(* CODESYS project XPlanar_Motion.library
   Author: Yuki
   Placeholder: XPlanar_Motion
   Title: XPlanar_Motion
   Version: 1.0
   DefaultNamespace: PM
   Company: Beckhoff

Project tree, tasks and I/O mapping:
  libraries: Tc2_MC2, * (Beckhoff Automation GmbH); Tc2_MC2_Camming, * (Beckhoff Automation GmbH); Tc2_Standard, * (Beckhoff Automation GmbH); Tc2_System, * (Beckhoff Automation GmbH); Tc3_Mc3PlanarMotion, * (Beckhoff Automation GmbH); Tc3_Module, * (Beckhoff Automation GmbH); Tc3_Physics, * (Beckhoff Automation GmbH); Tc3_XPlanarUtility, * (Beckhoff Automation GmbH & Co. KG)
  DUTs/
    data type ST_POSITION
  GVLs/
  POUs/
    General_FB/
      function block FB_StatusExecuteFB [ST]: METH_Busy, METH_CommandAborted, METH_Done, METH_Enter, METH_Error, METH_Execute, METH_Exit, METH_Main, Prop_Busy, Prop_CommandAborted, Prop_Done, Prop_Error, Prop_ErrorID, Prop_Execute
    Interface/
    MotionXPlanar/
      Basic/
        function block FB_Halt [ST]: METH_Busy, METH_Enter, METH_Exit, METH_Main
        function block FB_MoveA [ST]: METH_Busy, METH_Enter, METH_Exit, METH_Main
        function block FB_MoveB [ST]: METH_Busy, METH_Enter, METH_Exit, METH_Main
        function block FB_MoveC [ST]: METH_Busy, METH_Enter, METH_Exit, METH_Main
        function block FB_MoveToPosition [ST]: METH_Busy, METH_Enter, METH_Exit, METH_Main
        function block FB_MoveZ [ST]: METH_Busy, METH_Enter, METH_Exit, METH_Main
      Demo/
        function block FB_Corner [ST]: METH_Busy, METH_Enter, METH_Exit, METH_Main
        function block FB_ExternalSetPoint [ST]: ACT_SetExternalSetPoint, METH_Busy, METH_Enter, METH_Exit, METH_Main
        function block FB_Rotate_C [ST]: METH_Busy, METH_Enter, METH_Exit, METH_Main
        function block FB_Tilt_AB [ST]: METH_Busy, METH_Enter, METH_Exit, METH_Main
        function block FB_UpDown [ST]: METH_Busy, METH_Enter, METH_Exit, METH_Main
    ReadFB/
  VISUs/
*)

// DUTs/ST_POSITION
TYPE ST_POSITION :
STRUCT
	x					: LREAL;
	y					: LREAL;
	z					: LREAL;
	a					: LREAL;
	b					: LREAL;
	c					: LREAL;
END_STRUCT
END_TYPE

// POUs/General_FB/FB_StatusExecuteFB
 {attribute 'hide'}
FUNCTION_BLOCK ABSTRACT FB_StatusExecuteFB
VAR_INPUT
END_VAR
VAR_OUTPUT
END_VAR
VAR
	bExecute						: BOOL;
	bBusy							: BOOL;
	bCommandAborted					: BOOL;
	bDone							: BOOL;
	bError							: BOOL;
	udiErrorID						: UDINT;
END_VAR

//{warning 'add method implementation '}
METHOD ABSTRACT METH_Busy : BOOL
END_METHOD

//{warning 'add method implementation '}
METHOD PROTECTED METH_CommandAborted : BOOL
Prop_CommandAborted := TRUE;
Prop_Busy := FALSE;
END_METHOD

//{warning 'add method implementation '}
METHOD PROTECTED METH_Done : BOOL
Prop_Done := TRUE;
Prop_Busy := FALSE;
END_METHOD

METHOD ABSTRACT METH_Enter : BOOL
VAR_INPUT
END_VAR
END_METHOD

//{warning 'add method implementation '}
METHOD PROTECTED METH_Error : BOOL
Prop_Error := TRUE;
Prop_Busy := FALSE;
END_METHOD

//{warning 'add method implementation '}
METHOD PROTECTED METH_Execute : BOOL
Prop_Execute := TRUE;
Prop_Busy := TRUE;
END_METHOD

METHOD ABSTRACT METH_Exit : BOOL
VAR_INPUT
END_VAR
END_METHOD

METHOD ABSTRACT METH_Main : BOOL
VAR_INPUT
END_VAR
END_METHOD

{warning 'add property implementation'}
PROPERTY Prop_Busy : BOOL
GET
Prop_Busy := bBusy;
END_GET
SET
bBusy := Prop_Busy;
END_SET
END_PROPERTY

{warning 'add property implementation'}
PROPERTY Prop_CommandAborted : BOOL
GET
Prop_CommandAborted := bCommandAborted;
END_GET
SET
bCommandAborted := Prop_CommandAborted;
END_SET
END_PROPERTY

{warning 'add property implementation'}
PROPERTY Prop_Done : BOOL
GET
Prop_Done := bDone;
END_GET
SET
bDone := Prop_Done;
END_SET
END_PROPERTY

{warning 'add property implementation'}
PROPERTY Prop_Error : BOOL
GET
Prop_Error := bError;
END_GET
SET
bError := Prop_Error;
END_SET
END_PROPERTY

{warning 'add property implementation'}
PROPERTY Prop_ErrorID : UDINT
GET
Prop_ErrorID := udiErrorID;
END_GET
SET
udiErrorID := Prop_ErrorID;
END_SET
END_PROPERTY

{warning 'add property implementation'}
PROPERTY Prop_Execute : BOOL
GET
Prop_Execute := bExecute;
END_GET
SET
bExecute := Prop_Execute;
END_SET
END_PROPERTY

END_FUNCTION_BLOCK

// POUs/MotionXPlanar/Basic/FB_Halt
FUNCTION_BLOCK FB_Halt EXTENDS FB_StatusExecuteFB
VAR_IN_OUT
	fbMover								: MC_PlanarMover;
END_VAR
VAR_INPUT
	Execute								: BOOL;
	Velocity							: LREAL;
	Acceleration						: LREAL;
	Deceleration						: LREAL;
	Jerk								: LREAL;
END_VAR
VAR_OUTPUT
	Done								: BOOL;
	Busy								: BOOL;
	CommandAborted						: BOOL;
	Error								: BOOL;
	ErrorID								: UDINT;
END_VAR
VAR
	uiState								: UINT;
	//Input 内部変数
	lrVelocity							: LREAL;
	lrAcceleration						: LREAL;
	lrDeceleration						: LREAL;
	lrJerk								: LREAL;
	
	//ローカル
	fbFB_Mover							: MC_PlanarFeedback;
	fbConstraint						: DynamicConstraint_PathXY;
END_VAR

Prop_Execute := Execute;
METH_Main();
fbFB_Mover.Update();

Busy := bBusy;
Done := bDone;
CommandAborted := bCommandAborted;
Error := bError;
ErrorID := udiErrorID;

//{error 'add method implementation or delete method to use base implementation'}
METHOD METH_Busy : BOOL
IF fbFB_Mover.Error THEN
	METH_Error();
	Prop_ErrorID := fbFB_Mover.ErrorId; //Moverがエラー
	RETURN;
END_IF
IF THIS^.fbMover.MCTOPLC.STD.State = MC_PLANAR_STATE.Error THEN
	METH_Error();
	Prop_ErrorID := 1; //Moverがエラー
	RETURN;
END_IF
IF fbFB_Mover.Aborted THEN
	METH_CommandAborted();
	RETURN;
END_IF

CASE THIS^.uiState OF
	0:
	fbConstraint.SetValuesVADJ(V:= THIS^.lrVelocity, A:= THIS^.lrAcceleration, D:= THIS^.lrDeceleration, J:= THIS^.lrJerk);
	THIS^.fbMover.Halt(
		commandFeedback:= THIS^.fbFB_Mover, 
		constraint:= fbConstraint);

	THIS^.uiState := 10;	
	
	10:
	IF fbFB_Mover.Done THEN
		THIS^.uiState := 16#FFFF;	
	END_IF
	
	16#FFFF:
	METH_Done();
END_CASE
END_METHOD

//{error 'add method implementation or delete method to use base implementation'}
METHOD METH_Enter : BOOL
//Input 内部変数に移す
lrVelocity := Velocity;
lrAcceleration := Acceleration;
lrDeceleration := Deceleration;
lrJerk := Jerk;
END_METHOD

//{error 'add method implementation or delete method to use base implementation'}
METHOD METH_Exit : BOOL
Prop_Done := FALSE;
Prop_Busy := FALSE;
Prop_CommandAborted := FALSE;
Prop_Error := FALSE;
Prop_ErrorID := 0;

// 内部変数をリフレッシュする
uiState := 0;
lrVelocity := 0;
lrAcceleration := 0;
lrDeceleration := 0;
lrJerk := 0;
END_METHOD

//{error 'add method implementation or delete method to use base implementation'}
METHOD METH_Main : BOOL
//Doneに遷移
IF SUPER^.bDone AND SUPER^.bExecute THEN
	METH_Done();
	RETURN;
END_IF
//Errorに遷移
IF SUPER^.bError AND SUPER^.bExecute THEN
	METH_Error();
	RETURN;
END_IF
//CommandAbortedに遷移
IF SUPER^.bCommandAborted AND SUPER^.bExecute THEN
	METH_CommandAborted();
	RETURN;
END_IF
//FBをリフレッシュ
//状態がDone, Error, CommandAborted時に Execute FALSE で遷移
IF (SUPER^.bDone OR SUPER^.bError OR SUPER^.bCommandAborted) AND NOT SUPER^.bExecute THEN
	METH_Exit();
	RETURN;
END_IF

//実行開始
IF SUPER^.bExecute AND NOT SUPER^.bBusy THEN
	METH_Execute();
	METH_Enter();
END_IF
//実行中
IF SUPER^.bBusy THEN
	METH_Busy();
END_IF
END_METHOD

END_FUNCTION_BLOCK

// POUs/MotionXPlanar/Basic/FB_MoveA
FUNCTION_BLOCK FB_MoveA EXTENDS FB_StatusExecuteFB
VAR_IN_OUT
	fbMover								: MC_PlanarMover;
END_VAR
VAR_INPUT
	Execute								: BOOL;
	Position							: ST_POSITION;
	Velocity							: LREAL;
	Acceleration						: LREAL;
	Deceleration						: LREAL;
	Jerk								: LREAL;
END_VAR
VAR_OUTPUT
	Done								: BOOL;
	Busy								: BOOL;
	CommandAborted						: BOOL;
	Error								: BOOL;
	ErrorID								: UDINT;
END_VAR
VAR
	uiState								: UINT;
	//Input 内部変数
	dutPosition							: ST_POSITION;
	lrVelocity							: LREAL;
	lrAcceleration						: LREAL;
	lrDeceleration						: LREAL;
	lrJerk								: LREAL;
	
	//ローカル
	fbFB_Mover							: MC_PlanarFeedback;
	fbConstraint						: DynamicConstraint_PathXY;
END_VAR

Prop_Execute := Execute;
METH_Main();

fbFB_Mover.Update();

Busy := bBusy;
Done := bDone;
CommandAborted := bCommandAborted;
Error := bError;
ErrorID := udiErrorID;

//{error 'add method implementation or delete method to use base implementation'}
METHOD METH_Busy : BOOL
{warning disable C0371}
{warning restore C0371}
IF fbFB_Mover.Error THEN
	METH_Error();
	Prop_ErrorID := fbFB_Mover.ErrorId; //Moverがエラー
	RETURN;
END_IF
IF THIS^.fbMover.MCTOPLC.STD.State = MC_PLANAR_STATE.Error THEN
	METH_Error();
	Prop_ErrorID := 1; //Moverがエラー
	RETURN;
END_IF
IF fbFB_Mover.Aborted THEN
	METH_CommandAborted();
	RETURN;
END_IF

CASE THIS^.uiState OF
	0:
	fbConstraint.SetValuesVADJ(V:= THIS^.lrVelocity, A:= THIS^.lrAcceleration, D:= THIS^.lrDeceleration, J:= THIS^.lrJerk);
	THIS^.fbMover.MoveA(
		commandFeedback:= THIS^.fbFB_Mover, 
		targetPosition:= dutPosition.a, 
		constraint:= fbConstraint);

	THIS^.uiState := 10;	
	
	10:
	IF fbFB_Mover.Done THEN
		THIS^.uiState := 16#FFFF;	
	END_IF
	
	16#FFFF:
	METH_Done();
END_CASE
END_METHOD

//{error 'add method implementation or delete method to use base implementation'}
METHOD METH_Enter : BOOL
//Input 内部変数に移す
dutPosition := Position;
lrVelocity := Velocity;
lrAcceleration := Acceleration;
lrDeceleration := Deceleration;
lrJerk := Jerk;
END_METHOD

//{error 'add method implementation or delete method to use base implementation'}
METHOD METH_Exit : BOOL
Prop_Done := FALSE;
Prop_Busy := FALSE;
Prop_CommandAborted := FALSE;
Prop_Error := FALSE;
Prop_ErrorID := 0;

// 内部変数をリフレッシュする
uiState := 0;
lrVelocity := 0;
lrAcceleration := 0;
lrDeceleration := 0;
lrJerk := 0;
END_METHOD

//{error 'add method implementation or delete method to use base implementation'}
METHOD METH_Main : BOOL
//Doneに遷移
IF SUPER^.bDone AND SUPER^.bExecute THEN
	METH_Done();
	RETURN;
END_IF
//Errorに遷移
IF SUPER^.bError AND SUPER^.bExecute THEN
	METH_Error();
	RETURN;
END_IF
//CommandAbortedに遷移
IF SUPER^.bCommandAborted AND SUPER^.bExecute THEN
	METH_CommandAborted();
	RETURN;
END_IF
//FBをリフレッシュ
//状態がDone, Error, CommandAborted時に Execute FALSE で遷移
IF (SUPER^.bDone OR SUPER^.bError OR SUPER^.bCommandAborted) AND NOT SUPER^.bExecute THEN
	METH_Exit();
	RETURN;
END_IF

//実行開始
IF SUPER^.bExecute AND NOT SUPER^.bBusy THEN
	METH_Execute();
	METH_Enter();
END_IF
//実行中
IF SUPER^.bBusy THEN
	METH_Busy();
END_IF
END_METHOD

END_FUNCTION_BLOCK

// POUs/MotionXPlanar/Basic/FB_MoveB
FUNCTION_BLOCK FB_MoveB EXTENDS FB_StatusExecuteFB
VAR_IN_OUT
	fbMover								: MC_PlanarMover;
END_VAR
VAR_INPUT
	Execute								: BOOL;
	Position							: ST_POSITION;
	Velocity							: LREAL;
	Acceleration						: LREAL;
	Deceleration						: LREAL;
	Jerk								: LREAL;
END_VAR
VAR_OUTPUT
	Done								: BOOL;
	Busy								: BOOL;
	CommandAborted						: BOOL;
	Error								: BOOL;
	ErrorID								: UDINT;
END_VAR
VAR
	uiState								: UINT;
	//Input 内部変数
	dutPosition							: ST_POSITION;
	lrVelocity							: LREAL;
	lrAcceleration						: LREAL;
	lrDeceleration						: LREAL;
	lrJerk								: LREAL;
	
	//ローカル
	fbFB_Mover							: MC_PlanarFeedback;
	fbConstraint						: DynamicConstraint_PathXY;
END_VAR

Prop_Execute := Execute;
METH_Main();

fbFB_Mover.Update();

Busy := bBusy;
Done := bDone;
CommandAborted := bCommandAborted;
Error := bError;
ErrorID := udiErrorID;

//{error 'add method implementation or delete method to use base implementation'}
METHOD METH_Busy : BOOL
{warning disable C0371}
{warning restore C0371}
IF fbFB_Mover.Error THEN
	METH_Error();
	Prop_ErrorID := fbFB_Mover.ErrorId; //Moverがエラー
	RETURN;
END_IF
IF THIS^.fbMover.MCTOPLC.STD.State = MC_PLANAR_STATE.Error THEN
	METH_Error();
	Prop_ErrorID := 1; //Moverがエラー
	RETURN;
END_IF
IF fbFB_Mover.Aborted THEN
	METH_CommandAborted();
	RETURN;
END_IF

CASE THIS^.uiState OF
	0:
	fbConstraint.SetValuesVADJ(V:= THIS^.lrVelocity, A:= THIS^.lrAcceleration, D:= THIS^.lrDeceleration, J:= THIS^.lrJerk);
	THIS^.fbMover.MoveB(
		commandFeedback:= THIS^.fbFB_Mover, 
		targetPosition:= dutPosition.b, 
		constraint:= fbConstraint);

	THIS^.uiState := 10;	
	
	10:
	IF fbFB_Mover.Done THEN
		THIS^.uiState := 16#FFFF;	
	END_IF
	
	16#FFFF:
	METH_Done();
END_CASE
END_METHOD

//{error 'add method implementation or delete method to use base implementation'}
METHOD METH_Enter : BOOL
//Input 内部変数に移す
dutPosition := Position;
lrVelocity := Velocity;
lrAcceleration := Acceleration;
lrDeceleration := Deceleration;
lrJerk := Jerk;
END_METHOD

//{error 'add method implementation or delete method to use base implementation'}
METHOD METH_Exit : BOOL
Prop_Done := FALSE;
Prop_Busy := FALSE;
Prop_CommandAborted := FALSE;
Prop_Error := FALSE;
Prop_ErrorID := 0;

// 内部変数をリフレッシュする
uiState := 0;
lrVelocity := 0;
lrAcceleration := 0;
lrDeceleration := 0;
lrJerk := 0;
END_METHOD

//{error 'add method implementation or delete method to use base implementation'}
METHOD METH_Main : BOOL
//Doneに遷移
IF SUPER^.bDone AND SUPER^.bExecute THEN
	METH_Done();
	RETURN;
END_IF
//Errorに遷移
IF SUPER^.bError AND SUPER^.bExecute THEN
	METH_Error();
	RETURN;
END_IF
//CommandAbortedに遷移
IF SUPER^.bCommandAborted AND SUPER^.bExecute THEN
	METH_CommandAborted();
	RETURN;
END_IF
//FBをリフレッシュ
//状態がDone, Error, CommandAborted時に Execute FALSE で遷移
IF (SUPER^.bDone OR SUPER^.bError OR SUPER^.bCommandAborted) AND NOT SUPER^.bExecute THEN
	METH_Exit();
	RETURN;
END_IF

//実行開始
IF SUPER^.bExecute AND NOT SUPER^.bBusy THEN
	METH_Execute();
	METH_Enter();
END_IF
//実行中
IF SUPER^.bBusy THEN
	METH_Busy();
END_IF
END_METHOD

END_FUNCTION_BLOCK

// POUs/MotionXPlanar/Basic/FB_MoveC
FUNCTION_BLOCK FB_MoveC EXTENDS FB_StatusExecuteFB
VAR_IN_OUT
	fbMover								: MC_PlanarMover;
END_VAR
VAR_INPUT
	Execute								: BOOL;
	Position							: ST_POSITION;
	Velocity							: LREAL;
	Acceleration						: LREAL;
	Deceleration						: LREAL;
	Jerk								: LREAL;
END_VAR
VAR_OUTPUT
	Done								: BOOL;
	Busy								: BOOL;
	CommandAborted						: BOOL;
	Error								: BOOL;
	ErrorID								: UDINT;
END_VAR
VAR
	uiState								: UINT;
	//Input 内部変数
	dutPosition							: ST_POSITION;
	lrVelocity							: LREAL;
	lrAcceleration						: LREAL;
	lrDeceleration						: LREAL;
	lrJerk								: LREAL;
	
	//ローカル
	fbFB_Mover							: MC_PlanarFeedback;
	fbConstraint						: DynamicConstraint_PathXY;
	stMoveCOptions						: ST_MoveCOptions;
END_VAR

Prop_Execute := Execute;
METH_Main();

fbFB_Mover.Update();

Busy := bBusy;
Done := bDone;
CommandAborted := bCommandAborted;
Error := bError;
ErrorID := udiErrorID;

//{error 'add method implementation or delete method to use base implementation'}
METHOD METH_Busy : BOOL
IF fbFB_Mover.Error THEN
	METH_Error();
	Prop_ErrorID := fbFB_Mover.ErrorId; //Moverがエラー
	RETURN;
END_IF
IF THIS^.fbMover.MCTOPLC.STD.State = MC_PLANAR_STATE.Error THEN
	METH_Error();
	Prop_ErrorID := 1; //Moverがエラー
	RETURN;
END_IF
IF fbFB_Mover.Aborted THEN
	METH_CommandAborted();
	RETURN;
END_IF

CASE THIS^.uiState OF
	0:
	fbConstraint.SetValuesVADJ(V:= THIS^.lrVelocity, A:= THIS^.lrAcceleration, D:= THIS^.lrDeceleration, J:= THIS^.lrJerk);
	//ノンモジュロ設定有効
	stMoveCOptions.direction := Tc3_Mc3PlanarMotion.MC_DIRECTION.mcDirectionNonModulo;
	THIS^.fbMover.MoveC(
		commandFeedback:= THIS^.fbFB_Mover, 
		targetPosition:= dutPosition.c, 
		constraint:= fbConstraint, 
		options:= stMoveCOptions);
	THIS^.uiState := 10;	
	
	10:
	IF fbFB_Mover.Done THEN
		THIS^.uiState := 16#FFFF;	
	END_IF
	
	16#FFFF:
	METH_Done();
END_CASE
END_METHOD

//{error 'add method implementation or delete method to use base implementation'}
METHOD METH_Enter : BOOL
//Input 内部変数に移す
dutPosition := Position;
lrVelocity := Velocity;
lrAcceleration := Acceleration;
lrDeceleration := Deceleration;
lrJerk := Jerk;
END_METHOD

//{error 'add method implementation or delete method to use base implementation'}
METHOD METH_Exit : BOOL
Prop_Done := FALSE;
Prop_Busy := FALSE;
Prop_CommandAborted := FALSE;
Prop_Error := FALSE;
Prop_ErrorID := 0;

// 内部変数をリフレッシュする
uiState := 0;
lrVelocity := 0;
lrAcceleration := 0;
lrDeceleration := 0;
lrJerk := 0;
END_METHOD

//{error 'add method implementation or delete method to use base implementation'}
METHOD METH_Main : BOOL
//Doneに遷移
IF SUPER^.bDone AND SUPER^.bExecute THEN
	METH_Done();
	RETURN;
END_IF
//Errorに遷移
IF SUPER^.bError AND SUPER^.bExecute THEN
	METH_Error();
	RETURN;
END_IF
//CommandAbortedに遷移
IF SUPER^.bCommandAborted AND SUPER^.bExecute THEN
	METH_CommandAborted();
	RETURN;
END_IF
//FBをリフレッシュ
//状態がDone, Error, CommandAborted時に Execute FALSE で遷移
IF (SUPER^.bDone OR SUPER^.bError OR SUPER^.bCommandAborted) AND NOT SUPER^.bExecute THEN
	METH_Exit();
	RETURN;
END_IF

//実行開始
IF SUPER^.bExecute AND NOT SUPER^.bBusy THEN
	METH_Execute();
	METH_Enter();
END_IF
//実行中
IF SUPER^.bBusy THEN
	METH_Busy();
END_IF
END_METHOD

END_FUNCTION_BLOCK

// POUs/MotionXPlanar/Basic/FB_MoveToPosition
FUNCTION_BLOCK FB_MoveToPosition EXTENDS FB_StatusExecuteFB
VAR_IN_OUT
	fbMover								: MC_PlanarMover;
END_VAR
VAR_INPUT
	Execute								: BOOL;
	Position							: ST_POSITION;
	Velocity							: LREAL;
	Acceleration						: LREAL;
	Deceleration						: LREAL;
	Jerk								: LREAL;
END_VAR
VAR_OUTPUT
	Done								: BOOL;
	Busy								: BOOL;
	CommandAborted						: BOOL;
	Error								: BOOL;
	ErrorID								: UDINT;
END_VAR
VAR
	uiState								: UINT;
	//Input 内部変数
	xycPosition							: PositionXYC;
	dutPosition							: ST_POSITION;
	lrVelocity							: LREAL;
	lrAcceleration						: LREAL;
	lrDeceleration						: LREAL;
	lrJerk								: LREAL;
	
	//ローカル
	fbFB_Mover							: MC_PlanarFeedback;
	fbConstraint						: DynamicConstraint_PathXY;
END_VAR

Prop_Execute := Execute;
METH_Main();

fbFB_Mover.Update();

Busy := bBusy;
Done := bDone;
CommandAborted := bCommandAborted;
Error := bError;
ErrorID := udiErrorID;

//{warning 'add method implementation '}
//実行動作
METHOD METH_Busy : BOOL
IF fbFB_Mover.Error THEN
	METH_Error();
	Prop_ErrorID := fbFB_Mover.ErrorId; //Moverがエラー
	RETURN;
END_IF
IF THIS^.fbMover.MCTOPLC.STD.State = MC_PLANAR_STATE.Error THEN
	METH_Error();
	Prop_ErrorID := 1; //Moverがエラー
	RETURN;
END_IF
IF fbFB_Mover.Aborted THEN
	METH_CommandAborted();
	RETURN;
END_IF

CASE THIS^.uiState OF
	0:
	xycPosition.SetValuesXYC(x:= dutPosition.x, y:= dutPosition.y, c:= 0);
	fbConstraint.SetValuesVADJ(V:= THIS^.lrVelocity, A:= THIS^.lrAcceleration, D:= THIS^.lrDeceleration, J:= THIS^.lrJerk);
	THIS^.fbMover.MoveToPosition(
		commandFeedback:= THIS^.fbFB_Mover, 
		targetPosition:= xycPosition, 
		constraint:= fbConstraint, 
		options:= 0);
	THIS^.uiState := 10;
		
	10:
	IF fbFB_Mover.Done THEN
		THIS^.uiState := 16#FFFF;
	END_IF
	
	16#FFFF:
	METH_Done();
END_CASE
END_METHOD

METHOD METH_Enter : BOOL
VAR_INPUT
END_VAR
//Input 内部変数に移す
dutPosition := Position;
lrVelocity := Velocity;
lrAcceleration := Acceleration;
lrDeceleration := Deceleration;
lrJerk := Jerk;
END_METHOD

METHOD METH_Exit : BOOL
VAR_INPUT
END_VAR
Prop_Done := FALSE;
Prop_Busy := FALSE;
Prop_CommandAborted := FALSE;
Prop_Error := FALSE;
Prop_ErrorID := 0;

// 内部変数をリフレッシュする
uiState := 0;
xycPosition.SetValuesXYC(0,0,0);
lrVelocity := 0;
lrAcceleration := 0;
lrDeceleration := 0;
lrJerk := 0;
END_METHOD

METHOD METH_Main : BOOL
VAR_INPUT
END_VAR
//Doneに遷移
IF SUPER^.bDone AND SUPER^.bExecute THEN
	METH_Done();
	RETURN;
END_IF
//Errorに遷移
IF SUPER^.bError AND SUPER^.bExecute THEN
	METH_Error();
	RETURN;
END_IF
//CommandAbortedに遷移
IF SUPER^.bCommandAborted AND SUPER^.bExecute THEN
	METH_CommandAborted();
	RETURN;
END_IF
//FBをリフレッシュ
//状態がDone, Error, CommandAborted時に Execute FALSE で遷移
IF (SUPER^.bDone OR SUPER^.bError OR SUPER^.bCommandAborted) AND NOT SUPER^.bExecute THEN
	METH_Exit();
	RETURN;
END_IF

//実行開始
IF SUPER^.bExecute AND NOT SUPER^.bBusy THEN
	METH_Execute();
	METH_Enter();
END_IF
//実行中
IF SUPER^.bBusy THEN
	METH_Busy();
END_IF
END_METHOD

END_FUNCTION_BLOCK

// POUs/MotionXPlanar/Basic/FB_MoveZ
FUNCTION_BLOCK FB_MoveZ EXTENDS FB_StatusExecuteFB
VAR_IN_OUT
	fbMover								: MC_PlanarMover;
END_VAR
VAR_INPUT
	Execute								: BOOL;
	Position							: ST_POSITION;
	Velocity							: LREAL;
	Acceleration						: LREAL;
	Deceleration						: LREAL;
	Jerk								: LREAL;
END_VAR
VAR_OUTPUT
	Done								: BOOL;
	Busy								: BOOL;
	CommandAborted						: BOOL;
	Error								: BOOL;
	ErrorID								: UDINT;
END_VAR
VAR
	uiState								: UINT;
	//Input 内部変数
	dutPosition							: ST_POSITION;
	lrVelocity							: LREAL;
	lrAcceleration						: LREAL;
	lrDeceleration						: LREAL;
	lrJerk								: LREAL;
	
	//ローカル
	fbFB_Mover							: MC_PlanarFeedback;
	fbConstraint						: DynamicConstraint_PathXY;
END_VAR

Prop_Execute := Execute;
METH_Main();

fbFB_Mover.Update();

Busy := bBusy;
Done := bDone;
CommandAborted := bCommandAborted;
Error := bError;
ErrorID := udiErrorID;

//{error 'add method implementation or delete method to use base implementation'}
METHOD METH_Busy : BOOL
IF fbFB_Mover.Error THEN
	METH_Error();
	Prop_ErrorID := fbFB_Mover.ErrorId; //Moverがエラー
	RETURN;
END_IF
IF THIS^.fbMover.MCTOPLC.STD.State = MC_PLANAR_STATE.Error THEN
	METH_Error();
	Prop_ErrorID := 1; //Moverがエラー
	RETURN;
END_IF
IF fbFB_Mover.Aborted THEN
	METH_CommandAborted();
	RETURN;
END_IF

CASE THIS^.uiState OF
	0:
	fbConstraint.SetValuesVADJ(V:= THIS^.lrVelocity, A:= THIS^.lrAcceleration, D:= THIS^.lrDeceleration, J:= THIS^.lrJerk);
	THIS^.fbMover.MoveZ(
		commandFeedback:= THIS^.fbFB_Mover, 
		targetPosition:= dutPosition.z, 
		constraint:= fbConstraint);

	THIS^.uiState := 10;	
	
	10:
	IF fbFB_Mover.Done THEN
		THIS^.uiState := 16#FFFF;	
	END_IF
	
	16#FFFF:
	METH_Done();
END_CASE
END_METHOD

//{error 'add method implementation or delete method to use base implementation'}
METHOD METH_Enter : BOOL
//Input 内部変数に移す
dutPosition := Position;
lrVelocity := Velocity;
lrAcceleration := Acceleration;
lrDeceleration := Deceleration;
lrJerk := Jerk;
END_METHOD

//{error 'add method implementation or delete method to use base implementation'}
METHOD METH_Exit : BOOL
Prop_Done := FALSE;
Prop_Busy := FALSE;
Prop_CommandAborted := FALSE;
Prop_Error := FALSE;
Prop_ErrorID := 0;

// 内部変数をリフレッシュする
uiState := 0;
lrVelocity := 0;
lrAcceleration := 0;
lrDeceleration := 0;
lrJerk := 0;
END_METHOD

//{error 'add method implementation or delete method to use base implementation'}
METHOD METH_Main : BOOL
//Doneに遷移
IF SUPER^.bDone AND SUPER^.bExecute THEN
	METH_Done();
	RETURN;
END_IF
//Errorに遷移
IF SUPER^.bError AND SUPER^.bExecute THEN
	METH_Error();
	RETURN;
END_IF
//CommandAbortedに遷移
IF SUPER^.bCommandAborted AND SUPER^.bExecute THEN
	METH_CommandAborted();
	RETURN;
END_IF
//FBをリフレッシュ
//状態がDone, Error, CommandAborted時に Execute FALSE で遷移
IF (SUPER^.bDone OR SUPER^.bError OR SUPER^.bCommandAborted) AND NOT SUPER^.bExecute THEN
	METH_Exit();
	RETURN;
END_IF

//実行開始
IF SUPER^.bExecute AND NOT SUPER^.bBusy THEN
	METH_Execute();
	METH_Enter();
END_IF
//実行中
IF SUPER^.bBusy THEN
	METH_Busy();
END_IF
END_METHOD

END_FUNCTION_BLOCK

// POUs/MotionXPlanar/Demo/FB_Corner
FUNCTION_BLOCK FINAL FB_Corner EXTENDS FB_StatusExecuteFB
VAR_IN_OUT
	fbMover								: MC_PlanarMover;
END_VAR
VAR_INPUT
	Execute								: BOOL;
	Position							: ARRAY [0..3] OF ST_POSITION;
	Velocity							: LREAL;
	Acceleration						: LREAL;
	Deceleration						: LREAL;
	Jerk								: LREAL;
END_VAR
VAR_OUTPUT
	Done								: BOOL;
	Busy								: BOOL;
	CommandAborted						: BOOL;
	Error								: BOOL;
	ErrorID								: UDINT;
END_VAR
VAR
	uiState								: UINT;
	//Input 内部変数
	xycPosition							: PositionXYC;
	adutPosition							: ARRAY [0..3] OF ST_POSITION;
	lrVelocity							: LREAL;
	lrAcceleration						: LREAL;
	lrDeceleration						: LREAL;
	lrJerk								: LREAL;
	
	//ローカル
	fbFB_Mover							: MC_PlanarFeedback;
	fbMoveToPosition					: FB_MoveToPosition;
END_VAR

Prop_Execute := Execute;
METH_Main();

fbFB_Mover.Update();

Busy := bBusy;
Done := bDone;
CommandAborted := bCommandAborted;
Error := bError;
ErrorID := udiErrorID;

//{error 'add method implementation or delete method to use base implementation'}
METHOD METH_Busy : BOOL
{warning disable C0371}
{warning restore C0371}
IF fbFB_Mover.Error THEN
	METH_Error();
	Prop_ErrorID := fbFB_Mover.ErrorId; //Moverがエラー
	RETURN;
END_IF
IF THIS^.fbMover.MCTOPLC.STD.State = MC_PLANAR_STATE.Error THEN
	METH_Error();
	Prop_ErrorID := 1; //Moverがエラー
	RETURN;
END_IF
IF fbFB_Mover.Aborted THEN
	METH_CommandAborted();
	RETURN;
END_IF

CASE THIS^.uiState OF
	0:
	//配列0に移動
	fbMoveToPosition(
		fbMover:= THIS^.fbMover, 
		Execute:= TRUE, 
		Position:= adutPosition[0], 
		Velocity:= THIS^.lrVelocity, 
		Acceleration:= THIS^.lrAcceleration, 
		Deceleration:= THIS^.lrDeceleration, 
		Jerk:= THIS^.lrJerk);
	IF fbMoveToPosition.Done THEN
		fbMoveToPosition(fbMover:= THIS^.fbMover, Execute:= FALSE);
		THIS^.uiState := 10;
	ELSIF fbMoveToPosition.Error THEN
		METH_Error();
		Prop_ErrorID := 10; //Moverがエラー
	END_IF
	
	10:
	//配列1に動
	fbMoveToPosition(
		fbMover:= THIS^.fbMover, 
		Execute:= TRUE, 
		Position:= adutPosition[1], 
		Velocity:= THIS^.lrVelocity, 
		Acceleration:= THIS^.lrAcceleration, 
		Deceleration:= THIS^.lrDeceleration, 
		Jerk:= THIS^.lrJerk);
	IF fbMoveToPosition.Done THEN
		fbMoveToPosition(fbMover:= THIS^.fbMover, Execute:= FALSE);
		THIS^.uiState := 20;
	ELSIF fbMoveToPosition.Error THEN
		METH_Error();
		Prop_ErrorID := 11; //Moverがエラー
	END_IF
	
	20:
	//配列2に移動
	fbMoveToPosition(
		fbMover:= THIS^.fbMover, 
		Execute:= TRUE, 
		Position:= adutPosition[2], 
		Velocity:= THIS^.lrVelocity, 
		Acceleration:= THIS^.lrAcceleration, 
		Deceleration:= THIS^.lrDeceleration, 
		Jerk:= THIS^.lrJerk);
	IF fbMoveToPosition.Done THEN
		fbMoveToPosition(fbMover:= THIS^.fbMover, Execute:= FALSE);
		THIS^.uiState := 30;
	ELSIF fbMoveToPosition.Error THEN
		METH_Error();
		Prop_ErrorID := 13; //Moverがエラー
	END_IF
	
	30:
	//配列3に移動
	fbMoveToPosition(
		fbMover:= THIS^.fbMover, 
		Execute:= TRUE, 
		Position:= adutPosition[3], 
		Velocity:= THIS^.lrVelocity, 
		Acceleration:= THIS^.lrAcceleration, 
		Deceleration:= THIS^.lrDeceleration, 
		Jerk:= THIS^.lrJerk);
	IF fbMoveToPosition.Done THEN
		fbMoveToPosition(fbMover:= THIS^.fbMover, Execute:= FALSE);
		THIS^.uiState := 16#FFFF;
	ELSIF fbMoveToPosition.Error THEN
		METH_Error();
		Prop_ErrorID := 14; //Moverがエラー
	END_IF
	
	16#FFFF:
	METH_Done();
END_CASE
END_METHOD

 {attribute 'hide'}
//{error 'add method implementation or delete method to use base implementation'}
METHOD METH_Enter : BOOL
//Input 内部変数に移す
adutPosition := Position;
lrVelocity := Velocity;
lrAcceleration := Acceleration;
lrDeceleration := Deceleration;
lrJerk := Jerk;
END_METHOD

 {attribute 'hide'}
//{error 'add method implementation or delete method to use base implementation'}
METHOD METH_Exit : BOOL
Prop_Done := FALSE;
Prop_Busy := FALSE;
Prop_CommandAborted := FALSE;
Prop_Error := FALSE;
Prop_ErrorID := 0;

// 内部変数をリフレッシュする
uiState := 0;
xycPosition.SetValuesXYC(0,0,0);
lrVelocity := 0;
lrAcceleration := 0;
lrDeceleration := 0;
lrJerk := 0;

fbMoveToPosition(fbMover:= THIS^.fbMover, Execute:= FALSE);
END_METHOD

 {attribute 'hide'}
//{error 'add method implementation or delete method to use base implementation'}
METHOD METH_Main : BOOL
//Doneに遷移
IF SUPER^.bDone AND SUPER^.bExecute THEN
	METH_Done();
	RETURN;
END_IF
//Errorに遷移
IF SUPER^.bError AND SUPER^.bExecute THEN
	METH_Error();
	RETURN;
END_IF
//CommandAbortedに遷移
IF SUPER^.bCommandAborted AND SUPER^.bExecute THEN
	METH_CommandAborted();
	RETURN;
END_IF
//FBをリフレッシュ
//状態がDone, Error, CommandAborted時に Execute FALSE で遷移
IF (SUPER^.bDone OR SUPER^.bError OR SUPER^.bCommandAborted) AND NOT SUPER^.bExecute THEN
	METH_Exit();
	RETURN;
END_IF

//実行開始
IF SUPER^.bExecute AND NOT SUPER^.bBusy THEN
	METH_Execute();
	METH_Enter();
END_IF
//実行中
IF SUPER^.bBusy THEN
	METH_Busy();
END_IF
END_METHOD

END_FUNCTION_BLOCK

// POUs/MotionXPlanar/Demo/FB_ExternalSetPoint
FUNCTION_BLOCK FINAL FB_ExternalSetPoint EXTENDS FB_StatusExecuteFB
VAR_IN_OUT
	fbMover								: MC_PlanarMover;
	fbAxis_Master						: AXIS_REF;
	fbAxis_Slave_x						: AXIS_REF;
	fbAxis_Slave_y						: AXIS_REF;
	fbAxis_Slave_z						: AXIS_REF;
	fbAxis_Slave_a						: AXIS_REF;
	fbAxis_Slave_b						: AXIS_REF;
	fbAxis_Slave_c						: AXIS_REF;
END_VAR
VAR_INPUT
	Execute								: BOOL;
	Position							: ST_POSITION; //x: Master Position
	Velocity							: LREAL;
	Acceleration						: LREAL;
	Deceleration						: LREAL;
	Jerk								: LREAL;
END_VAR
VAR_OUTPUT
	Done								: BOOL;
	Busy								: BOOL;
	CommandAborted						: BOOL;
	Error								: BOOL;
	ErrorID								: UDINT;
END_VAR
VAR
	uiState								: UINT;
	//Input 内部変数
	dutPosition							: ST_POSITION;
	lrVelocity							: LREAL;
	lrAcceleration						: LREAL;
	lrDeceleration						: LREAL;
	lrJerk								: LREAL;
	
	//ローカル
	fbFB_Mover							: MC_PlanarFeedback;
	fbMoveZ								: FB_MoveZ;
	fbMoveB								: FB_MoveB;
	fbMoveToPosition					: FB_MoveToPosition;
	fbCamIn_S_x							: MC_CamIn;
	fbCamIn_S_y							: MC_CamIn;
	fbCamIn_S_a							: MC_CamIn;
	fbCamIn_S_b							: MC_CamIn;
	fbCamOut_S_x						: MC_CamOut;
	fbCamOut_S_y						: MC_CamOut;
	fbCamOut_S_a						: MC_CamOut;
	fbCamOut_S_b						: MC_CamOut;
	fbAbsolute_M						: MC_MoveAbsolute;
	stMoverVector_ActPos				: MoverVector;
	stMoverVector_ActVel				: MoverVector;
	stMoverVector_ActAcc				: MoverVector;
	dutTargetPosition					: ST_POSITION;
	bSetExternalSetPoint				: BOOL;
	stExternalOpt						: ST_ExternalSetpointGenerationOptions;
END_VAR

VAR CONSTANT
	//傾き量
	lrStrringStartPos_x					: LREAL := -40;
	lrStrringStartPos_z					: LREAL := 4;
	lrStrringStartPos_b					: LREAL := -2;
	lrStrringEndPos_z					: LREAL := 2;
	lrStrringEndPos_b					: LREAL := 0;
	
	//State
	State_StartPosition					: UINT := 0;
	State_StartZ						: UINT := 10;
	State_StartB						: UINT := 20;
	State_StartExternal					: UINT := 30;
	State_CamIn							: UINT := 40;
	State_StrringPlus					: UINT := 50;
	State_StrringMinus					: UINT := 60;
	State_EndExternal					: UINT := 70;
	State_CamOut						: UINT := 80;
	State_EndPosition					: UINT := 90;
	State_EndZ							: UINT := 100;
	State_EndB							: UINT := 110;
END_VAR

Prop_Execute := Execute;
METH_Main();

Busy := bBusy;
Done := bDone;
CommandAborted := bCommandAborted;
Error := bError;
ErrorID := udiErrorID;

ACTION ACT_SetExternalSetPoint:
stMoverVector_ActPos.x := THIS^.fbAxis_Slave_x.NcToPlc.ActPos;
stMoverVector_ActPos.y := THIS^.fbAxis_Slave_y.NcToPlc.ActPos;
stMoverVector_ActPos.z := THIS^.fbAxis_Slave_z.NcToPlc.ActPos;
stMoverVector_ActPos.a := THIS^.fbAxis_Slave_a.NcToPlc.ActPos;
stMoverVector_ActPos.b := THIS^.fbAxis_Slave_b.NcToPlc.ActPos;
stMoverVector_ActPos.c := THIS^.fbAxis_Slave_c.NcToPlc.ActPos;

stMoverVector_ActVel.x := THIS^.fbAxis_Slave_x.NcToPlc.ActVelo;
stMoverVector_ActVel.y := THIS^.fbAxis_Slave_y.NcToPlc.ActVelo;
stMoverVector_ActVel.z := THIS^.fbAxis_Slave_z.NcToPlc.ActVelo;
stMoverVector_ActVel.a := THIS^.fbAxis_Slave_a.NcToPlc.ActVelo;
stMoverVector_ActVel.b := THIS^.fbAxis_Slave_b.NcToPlc.ActVelo;
stMoverVector_ActVel.c := THIS^.fbAxis_Slave_c.NcToPlc.ActVelo;

stMoverVector_ActAcc.x := THIS^.fbAxis_Slave_x.NcToPlc.ActAcc;
stMoverVector_ActAcc.y := THIS^.fbAxis_Slave_y.NcToPlc.ActAcc;
stMoverVector_ActAcc.z := THIS^.fbAxis_Slave_z.NcToPlc.ActAcc;
stMoverVector_ActAcc.a := THIS^.fbAxis_Slave_a.NcToPlc.ActAcc;
stMoverVector_ActAcc.b := THIS^.fbAxis_Slave_b.NcToPlc.ActAcc;
stMoverVector_ActAcc.c := THIS^.fbAxis_Slave_c.NcToPlc.ActAcc;

THIS^.fbMover.SetExternalSetpoint(
	setPosition:= stMoverVector_ActPos, 
	setVelocity:= stMoverVector_ActVel, 
	setAcceleration:= stMoverVector_ActAcc);
END_ACTION

//{error 'add method implementation or delete method to use base implementation'}
METHOD METH_Busy : BOOL
{warning disable C0371}
{warning restore C0371}
IF fbFB_Mover.Error THEN
	METH_Error();
	Prop_ErrorID := fbFB_Mover.ErrorId; //Moverがエラー
	RETURN;
END_IF
IF THIS^.fbMover.MCTOPLC.STD.State = MC_PLANAR_STATE.Error THEN
	METH_Error();
	Prop_ErrorID := 1; //Moverがエラー
	RETURN;
END_IF
IF fbFB_Mover.Aborted THEN
	METH_CommandAborted();
	RETURN;
END_IF

IF bSetExternalSetPoint THEN
	ACT_SetExternalSetPoint();	
END_IF
CASE THIS^.uiState OF
	0:
	// ExternalSetpoint開始
	bSetExternalSetPoint := TRUE;
	stExternalOpt.mode := MC_EXTERNAL_SET_POSITION_MODE.Relative;
	THIS^.fbMover.StartExternalSetpointGeneration(commandFeedback:= 0, options:= stExternalOpt);
	THIS^.uiState := State_StrringPlus;
	
	State_StrringPlus: 
	//+360
	THIS^.fbAbsolute_M(
		Axis:= THIS^.fbAxis_Master, 
		Execute:= TRUE, 
		Position:= dutPosition.x, 
		Velocity:= THIS^.lrVelocity, 
		Acceleration:= THIS^.lrAcceleration, 
		Deceleration:= THIS^.lrDeceleration, 
		Jerk:= THIS^.lrJerk);
		
	IF THIS^.fbAbsolute_M.Done THEN
		THIS^.uiState := State_StrringMinus;
		THIS^.fbAbsolute_M(Axis:= THIS^.fbAxis_Master, Execute:= FALSE); 
	END_IF
	
	State_StrringMinus: 
	//原点に戻る
	THIS^.fbAbsolute_M(
		Axis:= THIS^.fbAxis_Master, 
		Execute:= TRUE, 
		Position:= 0, 
		Velocity:= THIS^.lrVelocity, 
		Acceleration:= THIS^.lrAcceleration, 
		Deceleration:= THIS^.lrDeceleration, 
		Jerk:= THIS^.lrJerk);
		
	IF THIS^.fbAbsolute_M.Done THEN
		THIS^.uiState := State_EndExternal;
		THIS^.fbAbsolute_M(Axis:= THIS^.fbAxis_Master, Execute:= FALSE); 
	END_IF
	
	State_EndExternal:
	// ExternalSetpoint終了
	bSetExternalSetPoint := FALSE;
	THIS^.fbMover.StopExternalSetpointGeneration(commandFeedback:= 0);
	THIS^.uiState := 16#FFFF;
	
	16#FFFF:
	METH_Done();
	
END_CASE

fbFB_Mover.Update();
END_METHOD

 {attribute 'hide'}
//{error 'add method implementation or delete method to use base implementation'}
METHOD METH_Enter : BOOL
//Input 内部変数に移す
dutPosition := Position;
lrVelocity := Velocity;
lrAcceleration := Acceleration;
lrDeceleration := Deceleration;
lrJerk := Jerk;
END_METHOD

 {attribute 'hide'}
//{error 'add method implementation or delete method to use base implementation'}
METHOD  METH_Exit : BOOL
Prop_Done := FALSE;
Prop_Busy := FALSE;
Prop_CommandAborted := FALSE;
Prop_Error := FALSE;
Prop_ErrorID := 0;

// 内部変数をリフレッシュする
uiState := 0;
lrVelocity := 0;
lrAcceleration := 0;
lrDeceleration := 0;
lrJerk := 0;
bSetExternalSetPoint :=FALSE;

//External Set Point 終了
THIS^.fbMover.StopExternalSetpointGeneration(commandFeedback:= 0);
END_METHOD

 {attribute 'hide'}
//{error 'add method implementation or delete method to use base implementation'}
METHOD METH_Main : BOOL
//Doneに遷移
IF SUPER^.bDone AND SUPER^.bExecute THEN
	METH_Done();
	RETURN;
END_IF
//Errorに遷移
IF SUPER^.bError AND SUPER^.bExecute THEN
	METH_Error();
	RETURN;
END_IF
//CommandAbortedに遷移
IF SUPER^.bCommandAborted AND SUPER^.bExecute THEN
	METH_CommandAborted();
	RETURN;
END_IF
//FBをリフレッシュ
//状態がDone, Error, CommandAborted時に Execute FALSE で遷移
IF (SUPER^.bDone OR SUPER^.bError OR SUPER^.bCommandAborted) AND NOT SUPER^.bExecute THEN
	METH_Exit();
	RETURN;
END_IF

//実行開始
IF SUPER^.bExecute AND NOT SUPER^.bBusy THEN
	METH_Execute();
	METH_Enter();
END_IF
//実行中
IF SUPER^.bBusy THEN
	METH_Busy();
END_IF
END_METHOD

END_FUNCTION_BLOCK

// POUs/MotionXPlanar/Demo/FB_Rotate_C
FUNCTION_BLOCK FINAL FB_Rotate_C EXTENDS FB_StatusExecuteFB
VAR_IN_OUT
	fbMover								: MC_PlanarMover;
END_VAR
VAR_INPUT
	Execute								: BOOL;
	Position							: ST_POSITION;
	Velocity							: LREAL;
	Acceleration						: LREAL;
	Deceleration						: LREAL;
	Jerk								: LREAL;
END_VAR
VAR_OUTPUT
	Done								: BOOL;
	Busy								: BOOL;
	CommandAborted						: BOOL;
	Error								: BOOL;
	ErrorID								: UDINT;
END_VAR
VAR
	uiState								: UINT;
	//Input 内部変数
	dutPosition							: ST_POSITION;
	lrVelocity							: LREAL;
	lrAcceleration						: LREAL;
	lrDeceleration						: LREAL;
	lrJerk								: LREAL;
	
	//ローカル
	fbFB_Mover							: MC_PlanarFeedback;
	dutTargetPosition					: ST_POSITION;
	fbConstraint						: DynamicConstraint_PathXY;
	fbMoveC								: FB_MoveC;
END_VAR

Prop_Execute := Execute;
METH_Main();

fbFB_Mover.Update();

Busy := bBusy;
Done := bDone;
CommandAborted := bCommandAborted;
Error := bError;
ErrorID := udiErrorID;

//{error 'add method implementation or delete method to use base implementation'}
METHOD METH_Busy : BOOL
IF fbFB_Mover.Error THEN
	METH_Error();
	Prop_ErrorID := fbFB_Mover.ErrorId; //Moverがエラー
	RETURN;
END_IF
IF THIS^.fbMover.MCTOPLC.STD.State = MC_PLANAR_STATE.Error THEN
	METH_Error();
	Prop_ErrorID := 1; //Moverがエラー
	RETURN;
END_IF
IF fbFB_Mover.Aborted THEN
	METH_CommandAborted();
	RETURN;
END_IF

CASE THIS^.uiState OF
	0:
	//+Cに回転
	dutTargetPosition.c := dutPosition.c;
	fbMoveC(
		fbMover:= THIS^.fbMover, 
		Execute:= TRUE, 
		Position:= dutTargetPosition, 
		Velocity:= THIS^.lrVelocity, 
		Acceleration:= THIS^.lrAcceleration, 
		Deceleration:= THIS^.lrDeceleration, 
		Jerk:= THIS^.lrJerk);
	IF fbMoveC.Done THEN
		fbMoveC(fbMover:= THIS^.fbMover, Execute:= FALSE);
		THIS^.uiState := 10;
	ELSIF fbMoveC.Error THEN
		METH_Error();
		Prop_ErrorID := 10; //Moverがエラー
	END_IF
	
	10:
	//-Cに回転
	dutTargetPosition.c := (-1)*dutPosition.c;
	fbMoveC(
		fbMover:= THIS^.fbMover, 
		Execute:= TRUE, 
		Position:= dutTargetPosition, 
		Velocity:= THIS^.lrVelocity, 
		Acceleration:= THIS^.lrAcceleration, 
		Deceleration:= THIS^.lrDeceleration, 
		Jerk:= THIS^.lrJerk);
	IF fbMoveC.Done THEN
		fbMoveC(fbMover:= THIS^.fbMover, Execute:= FALSE);
		THIS^.uiState := 20;
	ELSIF fbMoveC.Error THEN
		METH_Error();
		Prop_ErrorID := 11; //Moverがエラー
	END_IF
	
	20:
	//+Cに回転
	dutTargetPosition.c := 0;
	fbMoveC(
		fbMover:= THIS^.fbMover, 
		Execute:= TRUE, 
		Position:= dutTargetPosition, 
		Velocity:= THIS^.lrVelocity, 
		Acceleration:= THIS^.lrAcceleration, 
		Deceleration:= THIS^.lrDeceleration, 
		Jerk:= THIS^.lrJerk);
	IF fbMoveC.Done THEN
		fbMoveC(fbMover:= THIS^.fbMover, Execute:= FALSE);
		THIS^.uiState := 16#FFFF;
	ELSIF fbMoveC.Error THEN
		METH_Error();
		Prop_ErrorID := 12; //Moverがエラー
	END_IF
	
	16#FFFF:
	METH_Done();
END_CASE
END_METHOD

 {attribute 'hide'}
//{error 'add method implementation or delete method to use base implementation'}
METHOD METH_Enter : BOOL
//Input 内部変数に移す
dutPosition := Position;
lrVelocity := Velocity;
lrAcceleration := Acceleration;
lrDeceleration := Deceleration;
lrJerk := Jerk;
END_METHOD

 {attribute 'hide'}
//{error 'add method implementation or delete method to use base implementation'}
METHOD METH_Exit : BOOL
Prop_Done := FALSE;
Prop_Busy := FALSE;
Prop_CommandAborted := FALSE;
Prop_Error := FALSE;
Prop_ErrorID := 0;

// 内部変数をリフレッシュする
uiState := 0;
lrVelocity := 0;
lrAcceleration := 0;
lrDeceleration := 0;
lrJerk := 0;
END_METHOD

 {attribute 'hide'}
//{error 'add method implementation or delete method to use base implementation'}
METHOD METH_Main : BOOL
//Doneに遷移
IF SUPER^.bDone AND SUPER^.bExecute THEN
	METH_Done();
	RETURN;
END_IF
//Errorに遷移
IF SUPER^.bError AND SUPER^.bExecute THEN
	METH_Error();
	RETURN;
END_IF
//CommandAbortedに遷移
IF SUPER^.bCommandAborted AND SUPER^.bExecute THEN
	METH_CommandAborted();
	RETURN;
END_IF
//FBをリフレッシュ
//状態がDone, Error, CommandAborted時に Execute FALSE で遷移
IF (SUPER^.bDone OR SUPER^.bError OR SUPER^.bCommandAborted) AND NOT SUPER^.bExecute THEN
	METH_Exit();
	RETURN;
END_IF

//実行開始
IF SUPER^.bExecute AND NOT SUPER^.bBusy THEN
	METH_Execute();
	METH_Enter();
END_IF
//実行中
IF SUPER^.bBusy THEN
	METH_Busy();
END_IF
END_METHOD

END_FUNCTION_BLOCK

// POUs/MotionXPlanar/Demo/FB_Tilt_AB
FUNCTION_BLOCK FINAL FB_Tilt_AB EXTENDS FB_StatusExecuteFB
VAR_IN_OUT
	fbMover								: MC_PlanarMover;
END_VAR
VAR_INPUT
	Execute								: BOOL;
	Position							: ST_POSITION;
	Velocity							: LREAL;
	Acceleration						: LREAL;
	Deceleration						: LREAL;
	Jerk								: LREAL;
END_VAR
VAR_OUTPUT
	Done								: BOOL;
	Busy								: BOOL;
	CommandAborted						: BOOL;
	Error								: BOOL;
	ErrorID								: UDINT;
END_VAR
VAR
	uiState								: UINT;
	//Input 内部変数
	dutPosition							: ST_POSITION;
	lrVelocity							: LREAL;
	lrAcceleration						: LREAL;
	lrDeceleration						: LREAL;
	lrJerk								: LREAL;
	
	//ローカル
	fbFB_Mover							: MC_PlanarFeedback;
	dutTargetPosition					: ST_POSITION;
	fbConstraint						: DynamicConstraint_PathXY;
	fbMoveA								: FB_MoveA;
	fbMoveB								: FB_MoveB;
END_VAR

Prop_Execute := Execute;
METH_Main();

fbFB_Mover.Update();

Busy := bBusy;
Done := bDone;
CommandAborted := bCommandAborted;
Error := bError;
ErrorID := udiErrorID;

//{error 'add method implementation or delete method to use base implementation'}
METHOD METH_Busy : BOOL
IF fbFB_Mover.Error THEN
	METH_Error();
	Prop_ErrorID := fbFB_Mover.ErrorId; //Moverがエラー
	RETURN;
END_IF
IF THIS^.fbMover.MCTOPLC.STD.State = MC_PLANAR_STATE.Error THEN
	METH_Error();
	Prop_ErrorID := 1; //Moverがエラー
	RETURN;
END_IF
IF fbFB_Mover.Aborted THEN
	METH_CommandAborted();
	RETURN;
END_IF

CASE THIS^.uiState OF
	0:
	//+Aに傾ける
	dutTargetPosition.a := dutPosition.a;
	fbMoveA(
		fbMover:= THIS^.fbMover, 
		Execute:= TRUE, 
		Position:= dutTargetPosition, 
		Velocity:= THIS^.lrVelocity, 
		Acceleration:= THIS^.lrAcceleration, 
		Deceleration:= THIS^.lrDeceleration, 
		Jerk:= THIS^.lrJerk);
	IF fbMoveA.Done THEN
		fbMoveA(fbMover:= THIS^.fbMover, Execute:= FALSE);
		THIS^.uiState := 10;
	ELSIF fbMoveA.Error THEN
		METH_Error();
		Prop_ErrorID := 10; //Moverがエラー
	END_IF
	
	10:
	//+Bに傾ける
	dutTargetPosition.b := dutPosition.b;
	fbMoveB(
		fbMover:= THIS^.fbMover, 
		Execute:= TRUE, 
		Position:= dutTargetPosition, 
		Velocity:= THIS^.lrVelocity, 
		Acceleration:= THIS^.lrAcceleration, 
		Deceleration:= THIS^.lrDeceleration, 
		Jerk:= THIS^.lrJerk);
	IF fbMoveB.Done THEN
		fbMoveB(fbMover:= THIS^.fbMover, Execute:= FALSE);
		THIS^.uiState := 20;
	ELSIF fbMoveB.Error THEN
		METH_Error();
		Prop_ErrorID := 11; //Moverがエラー
	END_IF
	
	20:
	//-Aに傾ける
	dutTargetPosition.a := -1*dutPosition.a;
	fbMoveA(
		fbMover:= THIS^.fbMover, 
		Execute:= TRUE, 
		Position:= dutTargetPosition, 
		Velocity:= THIS^.lrVelocity, 
		Acceleration:= THIS^.lrAcceleration, 
		Deceleration:= THIS^.lrDeceleration, 
		Jerk:= THIS^.lrJerk);
	IF fbMoveA.Done THEN
		fbMoveA(fbMover:= THIS^.fbMover, Execute:= FALSE);
		THIS^.uiState := 30;
	ELSIF fbMoveA.Error THEN
		METH_Error();
		Prop_ErrorID := 12; //Moverがエラー
	END_IF
	
	30:
	//+Bに傾ける
	dutTargetPosition.b := -1*dutPosition.b;
	fbMoveB(
		fbMover:= THIS^.fbMover, 
		Execute:= TRUE, 
		Position:= dutTargetPosition, 
		Velocity:= THIS^.lrVelocity, 
		Acceleration:= THIS^.lrAcceleration, 
		Deceleration:= THIS^.lrDeceleration, 
		Jerk:= THIS^.lrJerk);
	IF fbMoveB.Done THEN
		fbMoveB(fbMover:= THIS^.fbMover, Execute:= FALSE);
		THIS^.uiState := 40;
	ELSIF fbMoveB.Error THEN
		METH_Error();
		Prop_ErrorID := 13; //Moverがエラー
	END_IF
	
	40:
	//0に戻す
	dutTargetPosition.a := 0;
	fbMoveA(
		fbMover:= THIS^.fbMover, 
		Execute:= TRUE, 
		Position:= dutTargetPosition, 
		Velocity:= THIS^.lrVelocity, 
		Acceleration:= THIS^.lrAcceleration, 
		Deceleration:= THIS^.lrDeceleration, 
		Jerk:= THIS^.lrJerk);
	IF fbMoveA.Done THEN
		fbMoveA(fbMover:= THIS^.fbMover, Execute:= FALSE);
		THIS^.uiState := 50;
	ELSIF fbMoveA.Error THEN
		METH_Error();
		Prop_ErrorID := 14; //Moverがエラー
	END_IF
	
	50:
	//0に戻す
	dutTargetPosition.b := 0;
	fbMoveB(
		fbMover:= THIS^.fbMover, 
		Execute:= TRUE, 
		Position:= dutTargetPosition, 
		Velocity:= THIS^.lrVelocity, 
		Acceleration:= THIS^.lrAcceleration, 
		Deceleration:= THIS^.lrDeceleration, 
		Jerk:= THIS^.lrJerk);
	IF fbMoveB.Done THEN
		fbMoveB(fbMover:= THIS^.fbMover, Execute:= FALSE);
		THIS^.uiState := 16#FFFF;
	ELSIF fbMoveB.Error THEN
		METH_Error();
		Prop_ErrorID := 15; //Moverがエラー
	END_IF
	
	16#FFFF:
	METH_Done();
END_CASE
END_METHOD

 {attribute 'hide'}
//{error 'add method implementation or delete method to use base implementation'}
METHOD METH_Enter : BOOL
//Input 内部変数に移す
dutPosition := Position;
lrVelocity := Velocity;
lrAcceleration := Acceleration;
lrDeceleration := Deceleration;
lrJerk := Jerk;
END_METHOD

 {attribute 'hide'}
//{error 'add method implementation or delete method to use base implementation'}
METHOD METH_Exit : BOOL
Prop_Done := FALSE;
Prop_Busy := FALSE;
Prop_CommandAborted := FALSE;
Prop_Error := FALSE;
Prop_ErrorID := 0;

// 内部変数をリフレッシュする
uiState := 0;
lrVelocity := 0;
lrAcceleration := 0;
lrDeceleration := 0;
lrJerk := 0;
END_METHOD

 {attribute 'hide'}
//{error 'add method implementation or delete method to use base implementation'}
METHOD METH_Main : BOOL
//Doneに遷移
IF SUPER^.bDone AND SUPER^.bExecute THEN
	METH_Done();
	RETURN;
END_IF
//Errorに遷移
IF SUPER^.bError AND SUPER^.bExecute THEN
	METH_Error();
	RETURN;
END_IF
//CommandAbortedに遷移
IF SUPER^.bCommandAborted AND SUPER^.bExecute THEN
	METH_CommandAborted();
	RETURN;
END_IF
//FBをリフレッシュ
//状態がDone, Error, CommandAborted時に Execute FALSE で遷移
IF (SUPER^.bDone OR SUPER^.bError OR SUPER^.bCommandAborted) AND NOT SUPER^.bExecute THEN
	METH_Exit();
	RETURN;
END_IF

//実行開始
IF SUPER^.bExecute AND NOT SUPER^.bBusy THEN
	METH_Execute();
	METH_Enter();
END_IF
//実行中
IF SUPER^.bBusy THEN
	METH_Busy();
END_IF
END_METHOD

END_FUNCTION_BLOCK

// POUs/MotionXPlanar/Demo/FB_UpDown
FUNCTION_BLOCK FINAL FB_UpDown EXTENDS FB_StatusExecuteFB
VAR_IN_OUT
	fbMover								: MC_PlanarMover;
END_VAR
VAR_INPUT
	Execute								: BOOL;
	Position							: ST_POSITION;
	Velocity							: LREAL;
	Acceleration						: LREAL;
	Deceleration						: LREAL;
	Jerk								: LREAL;
END_VAR
VAR_OUTPUT
	Done								: BOOL;
	Busy								: BOOL;
	CommandAborted						: BOOL;
	Error								: BOOL;
	ErrorID								: UDINT;
END_VAR
VAR
	uiState								: UINT;
	//Input 内部変数
	dutPosition							: ST_POSITION;
	lrVelocity							: LREAL;
	lrAcceleration						: LREAL;
	lrDeceleration						: LREAL;
	lrJerk								: LREAL;
	
	//ローカル
	fbFB_Mover							: MC_PlanarFeedback;
	dutTargetPosition					: ST_POSITION;
	fbConstraint						: DynamicConstraint_PathXY;
	fbMoveZ								: FB_MoveZ;
END_VAR

Prop_Execute := Execute;
METH_Main();

Busy := bBusy;
Done := bDone;
CommandAborted := bCommandAborted;
Error := bError;
ErrorID := udiErrorID;

//{error 'add method implementation or delete method to use base implementation'}
METHOD METH_Busy : BOOL
IF fbFB_Mover.Error THEN
	METH_Error();
	Prop_ErrorID := fbFB_Mover.ErrorId; //Moverがエラー
	RETURN;
END_IF
IF THIS^.fbMover.MCTOPLC.STD.State = MC_PLANAR_STATE.Error THEN
	METH_Error();
	Prop_ErrorID := 1; //Moverがエラー
	RETURN;
END_IF
IF fbFB_Mover.Aborted THEN
	METH_CommandAborted();
	RETURN;
END_IF

CASE THIS^.uiState OF
	0:
	//+Zに上昇
	dutTargetPosition.z := dutPosition.z;
	fbMoveZ(
		fbMover:= THIS^.fbMover, 
		Execute:= TRUE, 
		Position:= dutTargetPosition, 
		Velocity:= THIS^.lrVelocity, 
		Acceleration:= THIS^.lrAcceleration, 
		Deceleration:= THIS^.lrDeceleration, 
		Jerk:= THIS^.lrJerk);
	IF fbMoveZ.Done THEN
		fbMoveZ(fbMover:= THIS^.fbMover, Execute:= FALSE);
		THIS^.uiState := 10;
	ELSIF fbMoveZ.Error THEN
		METH_Error();
		Prop_ErrorID := 10; //Moverがエラー
	END_IF
	
	10:
	//ZにDefaultに設定
	dutTargetPosition.z := 2.0;
	fbMoveZ(
		fbMover:= THIS^.fbMover, 
		Execute:= TRUE, 
		Position:= dutTargetPosition, 
		Velocity:= THIS^.lrVelocity, 
		Acceleration:= THIS^.lrAcceleration, 
		Deceleration:= THIS^.lrDeceleration, 
		Jerk:= THIS^.lrJerk);
	IF fbMoveZ.Done THEN
		fbMoveZ(fbMover:= THIS^.fbMover, Execute:= FALSE);
		THIS^.uiState := 16#FFFF;
	ELSIF fbMoveZ.Error THEN
		METH_Error();
		Prop_ErrorID := 11; //Moverがエラー
	END_IF
	
	16#FFFF:
	METH_Done();
END_CASE

fbFB_Mover.Update();
END_METHOD

 {attribute 'hide'}
//{error 'add method implementation or delete method to use base implementation'}
METHOD METH_Enter : BOOL
//Input 内部変数に移す
dutPosition := Position;
lrVelocity := Velocity;
lrAcceleration := Acceleration;
lrDeceleration := Deceleration;
lrJerk := Jerk;
END_METHOD

 {attribute 'hide'}
//{error 'add method implementation or delete method to use base implementation'}
METHOD METH_Exit : BOOL
Prop_Done := FALSE;
Prop_Busy := FALSE;
Prop_CommandAborted := FALSE;
Prop_Error := FALSE;
Prop_ErrorID := 0;

// 内部変数をリフレッシュする
uiState := 0;
lrVelocity := 0;
lrAcceleration := 0;
lrDeceleration := 0;
lrJerk := 0;
END_METHOD

 {attribute 'hide'}
//{error 'add method implementation or delete method to use base implementation'}
METHOD METH_Main : BOOL
//Doneに遷移
IF SUPER^.bDone AND SUPER^.bExecute THEN
	METH_Done();
	RETURN;
END_IF
//Errorに遷移
IF SUPER^.bError AND SUPER^.bExecute THEN
	METH_Error();
	RETURN;
END_IF
//CommandAbortedに遷移
IF SUPER^.bCommandAborted AND SUPER^.bExecute THEN
	METH_CommandAborted();
	RETURN;
END_IF
//FBをリフレッシュ
//状態がDone, Error, CommandAborted時に Execute FALSE で遷移
IF (SUPER^.bDone OR SUPER^.bError OR SUPER^.bCommandAborted) AND NOT SUPER^.bExecute THEN
	METH_Exit();
	RETURN;
END_IF

//実行開始
IF SUPER^.bExecute AND NOT SUPER^.bBusy THEN
	METH_Execute();
	METH_Enter();
END_IF
//実行中
IF SUPER^.bBusy THEN
	METH_Busy();
END_IF
END_METHOD

END_FUNCTION_BLOCK
